// TIA Portal V20 export
TYPE "zp_CITITradeCalls"
// stored: Namespace CITI_Logic
   STRUCT
      Call_1 : Bool;   // Trade Call 1
      Call_2 : Bool;   // Trade Call 2
      Call_3 : Bool;   // Trade Call 3
      Call_4 : Bool;   // Trade Call 4
      Call_5 : Bool;   // Trade Call 5
      Call_6 : Bool;   // Trade Call 6
      Call_7 : Bool;   // Trade Call 7
      Call_8 : Bool;   // Trade Call 8
      CallAck_1 : Bool;   // Trade Call Acknowledge 1
      CallAck_2 : Bool;   // Trade Call Acknowledge 2
      CallAck_3 : Bool;   // Trade Call Acknowledge 3
      CallAck_4 : Bool;   // Trade Call Acknowledge 4
      CallAck_5 : Bool;   // Trade Call Acknowledge 5
      CallAck_6 : Bool;   // Trade Call Acknowledge 6
      CallAck_7 : Bool;   // Trade Call Acknowledge 7
      CallAck_8 : Bool;   // Trade Call Acknowledge 8
   END_STRUCT;
END_TYPE
